Universal Robots PolyScope program: square_motion_relative_to_the_tool_with_blends.urp

ProgramRoot directory=/home/esben/programs; name=square_motion_relative_to_the_tool_with_blends; robotEnvironmentFileName=default
  MainProgram cartesianAcceleration=1.2; cartesianSpeed=0.25; jointAcceleration=1.3962634015954636; jointSpeed=1.0471975511965976; moveAsFastAsPossible=true; motionType=JOINT_SPACE
    Assignment assignmentValueSource=0; expr=get_forward_kin(); operatorValueType=INTEGER; valueSource=EXPRESSION; variable=(name=start_pos, prefersPersistentValue=false, requestANewUniqueName=false)
    Assignment assignmentValueSource=0; assignmentOperatorMessage=Height in mm?; operatorValueType=FLOAT; valueSource=OPERATOR; variable=(name=height, prefersPersistentValue=false, requestANewUniqueName=false)
    Assignment assignmentValueSource=0; assignmentOperatorMessage=Width in mm?; operatorValueType=FLOAT; valueSource=OPERATOR; variable=(name=width, prefersPersistentValue=false, requestANewUniqueName=false)
    While count=0; type=LOOP_FOREVER; variable=(name=Loop, prefersPersistentValue=false, requestANewUniqueName=true)
      Move cartesianAcceleration=1.2; cartesianSpeed=0.25; jointAcceleration=1.3962634015954636; jointSpeed=1.0471975511965976; moveAsFastAsPossible=true; motionType=CARTESIAN_SPACE
        Assignment assignmentValueSource=0; assignmentOperatorMessage=pose_trans(start_pos,p[width/1000.0,0.0,0.0,0.0,0.0,0.0]); expr=pose_trans(start_pos,p[ExpressionVariableNode/1000.0,0.0,0.0,0.0,0.0,0.0]); operatorValueType=INTEGER; valueSource=EXPRESSION; variable=(name=corner_1, prefersPersistentValue=false, requestANewUniqueName=false)
        Waypoint blendRadius=0.05; cartesianAcceleration=1.2; cartesianSpeed=0.25; jointAcceleration=1.3962634015954636; jointSpeed=1.0471975511965976; nextMotionTime=2.0; useSharedParameters=true; positionType=VARIABLE_POSITION; variable=(name=corner_1, prefersPersistentValue=false, requestANewUniqueName=false); name=Waypoint
      Move cartesianAcceleration=1.2; cartesianSpeed=0.25; jointAcceleration=1.3962634015954636; jointSpeed=1.0471975511965976; moveAsFastAsPossible=true; motionType=CARTESIAN_SPACE
        Assignment assignmentValueSource=0; expr=pose_trans(start_pos,p[width/1000.0,height/1000.0,0.0,0.0,0.0,0.0]); operatorValueType=INTEGER; valueSource=EXPRESSION; variable=(name=corner_2, prefersPersistentValue=false, requestANewUniqueName=false)
        Waypoint blendRadius=0.05; cartesianAcceleration=1.2; cartesianSpeed=0.25; jointAcceleration=1.3962634015954636; jointSpeed=1.0471975511965976; nextMotionTime=2.0; useSharedParameters=true; positionType=VARIABLE_POSITION; variable=(name=corner_2, prefersPersistentValue=false, requestANewUniqueName=false); name=Waypoint
      Move cartesianAcceleration=1.2; cartesianSpeed=0.25; jointAcceleration=1.3962634015954636; jointSpeed=1.0471975511965976; moveAsFastAsPossible=true; motionType=CARTESIAN_SPACE
        Assignment assignmentValueSource=0; assignmentOperatorMessage=pose_trans(p[0.0,hieght/1000.0,0.0,0.0,0.0,0.0],start_pos); expr=pose_trans(start_pos,p[0.0,height/1000.0,0.0,0.0,0.0,0.0]); operatorValueType=INTEGER; valueSource=EXPRESSION; variable=(name=corner_3, prefersPersistentValue=false, requestANewUniqueName=false)
        Waypoint blendRadius=0.05; cartesianAcceleration=1.2; cartesianSpeed=0.25; jointAcceleration=1.3962634015954636; jointSpeed=1.0471975511965976; nextMotionTime=2.0; useSharedParameters=true; positionType=VARIABLE_POSITION; variable=(name=corner_3, prefersPersistentValue=false, requestANewUniqueName=false); name=Waypoint
      Move cartesianAcceleration=1.2; cartesianSpeed=0.25; jointAcceleration=1.3962634015954636; jointSpeed=1.0471975511965976; moveAsFastAsPossible=true; motionType=CARTESIAN_SPACE
        Waypoint blendRadius=0.05; cartesianAcceleration=1.2; cartesianSpeed=0.25; jointAcceleration=1.3962634015954636; jointSpeed=1.0471975511965976; nextMotionTime=2.0; useSharedParameters=true; positionType=VARIABLE_POSITION; variable=(name=start_pos, prefersPersistentValue=false, requestANewUniqueName=false); name=Waypoint
